(*
SPDX-FileCopyrightText: © 2026 Oleksandr Tiutyk <trofimich@gmail.com>
SPDX-License-Identifier: MIT
License: https://opensource.org/license/mit
*)

(*!
<summary>Receives the library namespace through compiler initialization.</summary>
<description>
CurrentNamespace is metadata storage; callers borrow it read-only through CurrentNamespace.Name.
</description>
*)

FUNCTION_BLOCK INTERNAL NamespaceExtractor
VAR_OUTPUT
	{attribute 'init_namespace'} 
	CurrentNamespace : STRING; 	
END_VAR

END_FUNCTION_BLOCK

(* stored: Version 1.1.0.1
   POU NamespaceExtractor: Id {775a0944-5518-486b-9fd6-59adf0116bbf}, SpecialFunc None *)
